Yaskawa INFORM job: R1_W68-69(-90,-90)KM-OK-R2.JBI

/JOB
//NAME R1_W68-69(-90,-90)KM-OK-R2
///FOLDERNAME KRIS-SCIANA
//POS
///NPOS 38,38,0,3,0,0
///TOOL 0
///POSTYPE PULSE
///PULSE
C00000=73468,9895,-28016,-5981,91523,26793
C00001=120734,71276,72201,4504,87810,-53709
C00002=120735,71272,72196,4504,87811,-53709
C00003=121395,68528,69777,4569,87853,-53485
C00004=121395,69171,71254,4570,87276,-53507
C00005=121395,68528,69777,4569,87853,-53485
C00006=121401,65302,66136,4570,88433,-53462
C00007=121395,68528,69777,4569,87853,-53485
C00008=112016,77626,86184,20885,85648,-58358
C00009=112809,77066,85486,20996,85583,-58090
C00010=112016,77626,86184,20885,85648,-58358
C00011=120735,71328,72263,-1559,94817,-55545
C00012=120734,71336,72273,-1559,94815,-55545
C00013=120751,61561,41578,27514,97921,23508
C00014=120734,70951,71810,-2171,75229,66298
C00015=120734,70920,71772,-2171,75236,66298
C00016=121246,68263,69691,-2208,75166,66476
C00017=121246,68876,71092,-2211,74617,66486
C00018=121246,68263,69691,-2208,75166,66476
C00019=121249,66081,67311,-2190,75512,66471
C00020=121246,68263,69691,-2208,75166,66476
C00021=118877,68193,69204,-2033,75369,65652
C00022=118283,68515,69855,-1990,75118,65451
C00023=118877,68193,69204,-2033,75369,65652
C00024=120734,70827,71660,4347,82001,67463
C00025=120734,70853,71692,4347,81995,67463
C00026=112400,61296,37228,-23103,109629,-28450
C00027=107341,71278,72203,-37113,101922,-81721
C00028=107341,71251,72171,-37114,101927,-81723
C00029=84385,41965,23634,1765,100233,-86576
C00030=107467,74944,76649,-36953,101288,-81446
C00031=107434,72961,73317,-37117,102107,-81746
C00032=101885,24330,30379,11380,107837,-79029
C00033=134483,20711,26868,21376,101470,-67962
C00034=126490,11045,23545,35813,94957,-73666
C00035=109663,20975,-134,16743,105523,-76722
C00036=109630,25453,-16548,18427,117386,-74878
C00037=-3257,25453,-16548,18427,77795,-74692
BC00000=44418,459057,864722
BC00001=87328,510185,591893
BC00002=84135,512442,568566
BC00003=82858,513344,559235
BC00004=82858,513344,559235
BC00005=82858,513344,559235
BC00006=82858,513344,559235
BC00007=82858,513344,559235
BC00008=82858,513344,559235
BC00009=82858,513344,559235
BC00010=82858,513344,559235
BC00011=71596,502428,561564
BC00012=73933,499123,584513
BC00013=161167,522419,507004
BC00014=155724,532187,604802
BC00015=157686,533891,579439
BC00016=158471,534573,569294
BC00017=158471,534573,569294
BC00018=158471,534573,569294
BC00019=158471,534573,569291
BC00020=158471,534573,569294
BC00021=158471,534573,569294
BC00022=158471,534573,569294
BC00023=158471,534573,569294
BC00024=176188,518019,576780
BC00025=175193,515360,601776
BC00026=108792,485533,523388
BC00027=68701,467524,476059
BC00028=71515,473252,460875
BC00029=72469,475194,455726
BC00030=72640,475543,454802
BC00031=72640,475543,454802
BC00032=140452,436459,555514
BC00033=140385,436497,555415
BC00034=140385,436497,555415
BC00035=72469,475194,455727
BC00036=72469,475193,455723
BC00037=72469,475193,748163
///POSTYPE BASE
///RECTAN
///RCONF 0,0,0,0,1,0,0,0,0,0,0,0,0,0,0,0,0,0,0,0,0,0,0,0
P00006=2.006,1.622,-0.565,0.0000,0.0000,0.0000
P00021=0.073,2.058,-0.109,0.0000,0.0000,0.0000
P00022=2.006,1.622,-0.565,0.0000,0.0000,0.0000
//INST
///DATE 2025/04/14 13:48
///ATTR SC,RW
///GROUP1 RB1,BS1
NOP
SFTOF
MOVJ C00000 BC00000 VJ=100.00
MOVJ C00001 BC00001 VJ=100.00
MOVL C00002 BC00002 V=100.0
MOVL C00003 BC00003 V=60.0
REFP 3 C00004 BC00004
CALL JOB:SEARCH-R1
SET P021 P006
SFTON P021
MOVL C00005 BC00005 V=60.0
REFP 3 C00006 BC00006
CALL JOB:SEARCH-R1
SET P021 P006
SFTON P021
MOVL C00007 BC00007 V=60.0
MOVL C00008 BC00008 V=60.0
REFP 3 C00009 BC00009
CALL JOB:SEARCH-R1
SET P021 P006
SFTON P021
MOVL C00010 BC00010 V=60.0
MOVL C00011 BC00011 V=100.0
MOVL C00012 BC00012 V=166.7
'Path VIA1138
SFTOF
MOVJ C00013 BC00013 VJ=100.00
'Path S759 (for W102)
SFTOF
MOVJ C00014 BC00014 VJ=100.00
MOVL C00015 BC00015 V=100.0
MOVL C00016 BC00016 V=60.0
REFP 3 C00017 BC00017
CALL JOB:SEARCH-R1
SET P022 P006
SFTON P022
MOVL C00018 BC00018 V=60.0
REFP 3 C00019 BC00019
CALL JOB:SEARCH-R1
SET P022 P006
SFTON P022
MOVL C00020 BC00020 V=60.0
MOVL C00021 BC00021 V=60.0
REFP 3 C00022 BC00022
CALL JOB:SEARCH-R1
SET P022 P006
SFTON P022
MOVL C00023 BC00023 V=60.0
MOVL C00024 BC00024 V=166.7
MOVL C00025 BC00025 V=166.7
'Path VIA1139
SFTOF
MOVJ C00026 BC00026 VJ=100.00
'Path W102
SFTOF
SFTON P022
CALL JOB:COFNIJ_DRUT
MOVJ C00027 BC00027 VJ=100.00
MOVL C00028 BC00028 V=166.7
MOVL C00029 BC00029 V=100.0 PL=0
REFP 1 C00030 BC00030
REFP 2 C00031 BC00031
MACRO1 MJ#(0) ARGF9
ARCON
MOVL C00032 BC00032 V=10.8
SFTON P021
MOVL C00033 BC00033 V=10.8
MOVL C00034 BC00034 V=10.8
ARCOF
MOVL C00035 BC00035 V=100.0
SFTOF
MOVJ C00036 BC00036 VJ=100.00
MOVJ C00037 BC00037 VJ=100.00
END
